TYPE ST_AlarmEntry :
STRUCT
	sTimestamp   : STRING(23);
	eSeverity    : E_AlarmSeverity;
	sMessage     : STRING(255);
	bActive      : BOOL;
END_STRUCT
END_TYPE

(* stored: Version 1.1.0.1, ProductVersion 3.1.4026.17
   DUT ST_AlarmEntry: Id {9b9bba10-6518-49bb-83f1-85f705052d69} *)
